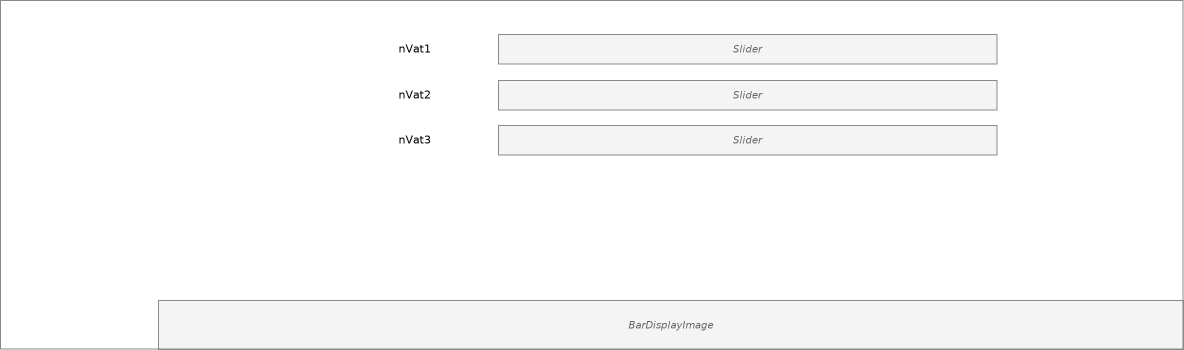
VISUALIZATION Visu  // 1184x350
    Slider (498,34 499x30), variable: MAIN.nVat1, scale 0..2000
    Slider (498,80 499x30), variable: MAIN.nVat2, scale 0..3000
    Slider (498,125 499x30), variable: MAIN.nVat3, scale 0..5000
    Label (340,34 150x30), "nVat1"
    Label (340,80 150x30), "nVat2"
    Label (340,125 150x30), "nVat3"
    BarDisplayImage (158,300 1026x50), value: MAIN.nTotaal, style: BarDisplayImage-Gray, scale format: %.1f, scale 0..10000
END_VISUALIZATION

(* stored: Version 1.1.0.1, ProductVersion 3.1.4024.12
   Visu Visu: Id {36e26788-c5e1-4c7a-8d95-03db61388b44} *)
